(* Logix 5000 project; controller FRC_CC_2020 vendor 1 type 14 code 150 rev 31.11; software revision 31.01; part 2 of 4 *)
(* tags used below, declared in another part *)
   BlueESTOP1 : ALIAS FOR Blue_Driver_station:I.Data.14;
   BlueESTOP2 : ALIAS FOR Blue_Driver_station:I.Data.12;
   BlueESTOP3 : ALIAS FOR Blue_Driver_station:I.Data.10;
   Connection : INT;
   Field_Reset_Green : BOOL;
   FieldESTOP : BOOL;
   FieldESTOPButton : ALIAS FOR Local:1:I.Data.0;
   MatchReset : BOOL;
   MatchSYNC : TIMER;
   MBTI_Change_Log_MSG : MESSAGE;
   MBTI_Conn_Acc_Timeout_MSG : MESSAGE;
   MBTI_Conn_Accept_MSG : MESSAGE;
   MBTI_ConnectionsLastErrors : DINT;
   MBTI_Create_Sock_MSG : MESSAGE;
   MBTI_Delete_All_MSG : MESSAGE;
   MBTI_Instance : DINT;
   MBTI_Read_Data_MSG_00 : MESSAGE;
   MBTI_Read_Data_MSG_01 : MESSAGE;
   MBTI_Read_Data_MSG_02 : MESSAGE;
   MBTI_Read_Data_MSG_03 : MESSAGE;
   MBTI_Read_Data_MSG_04 : MESSAGE;
   MBTI_Read_Data_MSG_05 : MESSAGE;
   MBTI_Read_Data_MSG_06 : MESSAGE;
   MBTI_Read_Data_MSG_07 : MESSAGE;
   MBTI_Read_Data_MSG_08 : MESSAGE;
   MBTI_Read_Data_MSG_09 : MESSAGE;
   MBTI_Read_Done : BOOL[32];
   MBTI_Read_Resp : READ_RESP_STR[10];
   MBTI_RW_Inactivity_MSG : MESSAGE;
   MBTI_Sock_Accept_Resp : AcceptResponse;
   MBTI_Total_Open : INT;
   MBTI_Total_Open_MSG : MESSAGE;
   MBTI_Write_Data_MSG_00 : MESSAGE;
   MBTI_Write_Data_MSG_01 : MESSAGE;
   MBTI_Write_Data_MSG_02 : MESSAGE;
   MBTI_Write_Data_MSG_03 : MESSAGE;
   MBTI_Write_Data_MSG_04 : MESSAGE;
   MBTI_Write_Data_MSG_05 : MESSAGE;
   MBTI_Write_Data_MSG_06 : MESSAGE;
   MBTI_Write_Data_MSG_07 : MESSAGE;
   MBTI_Write_Data_MSG_08 : MESSAGE;
   MBTI_Write_Data_MSG_09 : MESSAGE;
   MBTI_Write_Data_Out : WRT_DATA[10];
   MBTU_Enable_MBTCP : BOOL;
   MBTU_EnetModulePort : STRING;
   MBTU_Log_Enable : DINT;
   MBTU_MB_0xx : BOOL[256];
   MBTU_MB_1xx : BOOL[256];
   MBTU_MB_3xx : INT[1000];
   MBTU_MB_4xx : INT[100];
   RedESTOP1 : ALIAS FOR Red_Driver_station:I.Data.14;
   RedESTOP2 : ALIAS FOR Red_Driver_station:I.Data.12;
   RedESTOP3 : ALIAS FOR Red_Driver_station:I.Data.10;
   SL_1 : BOOL;
   SL_2 : BOOL;
   SL_3 : BOOL;
   SL_B : BOOL;
   Stack_Light_Green : ALIAS FOR Local:1:O.Data.4;
   Watchdog : BOOL;
(* MainProgram, continued *)

ROUTINE Tag_Converter_Static   (* ladder *)
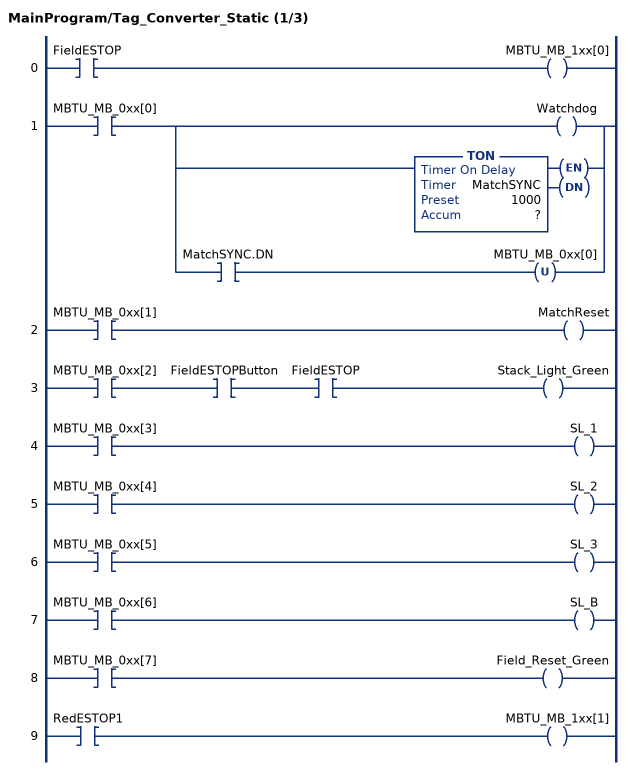
   0: XIC(FieldESTOP)OTE(MBTU_MB_1xx[0]);
   1: XIC(MBTU_MB_0xx[0])[OTE(Watchdog) ,TON(MatchSYNC,?,?) ,XIC(MatchSYNC.DN) OTU(MBTU_MB_0xx[0]) ];
   2: XIC(MBTU_MB_0xx[1])OTE(MatchReset);
   3: XIC(MBTU_MB_0xx[2])XIC(FieldESTOPButton)XIC(FieldESTOP)OTE(Stack_Light_Green);
   4: XIC(MBTU_MB_0xx[3])OTE(SL_1);
   5: XIC(MBTU_MB_0xx[4])OTE(SL_2);
   6: XIC(MBTU_MB_0xx[5])OTE(SL_3);
   7: XIC(MBTU_MB_0xx[6])OTE(SL_B);
   8: XIC(MBTU_MB_0xx[7])OTE(Field_Reset_Green);
   9: XIC(RedESTOP1)OTE(MBTU_MB_1xx[1]);
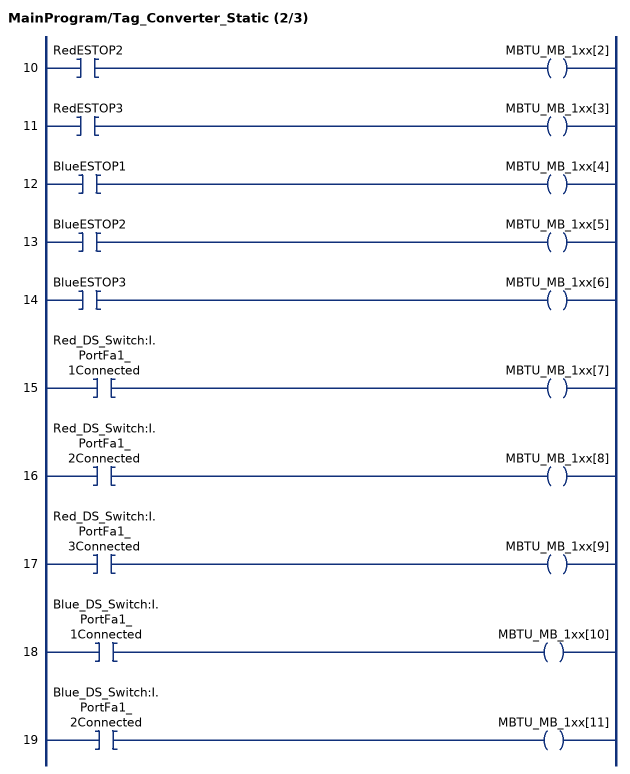
   10: XIC(RedESTOP2)OTE(MBTU_MB_1xx[2]);
   11: XIC(RedESTOP3)OTE(MBTU_MB_1xx[3]);
   12: XIC(BlueESTOP1)OTE(MBTU_MB_1xx[4]);
   13: XIC(BlueESTOP2)OTE(MBTU_MB_1xx[5]);
   14: XIC(BlueESTOP3)OTE(MBTU_MB_1xx[6]);
   15: XIC(Red_DS_Switch:I.PortFa1_1Connected)OTE(MBTU_MB_1xx[7]);
   16: XIC(Red_DS_Switch:I.PortFa1_2Connected)OTE(MBTU_MB_1xx[8]);
   17: XIC(Red_DS_Switch:I.PortFa1_3Connected)OTE(MBTU_MB_1xx[9]);
   18: XIC(Blue_DS_Switch:I.PortFa1_1Connected)OTE(MBTU_MB_1xx[10]);
   19: XIC(Blue_DS_Switch:I.PortFa1_2Connected)OTE(MBTU_MB_1xx[11]);
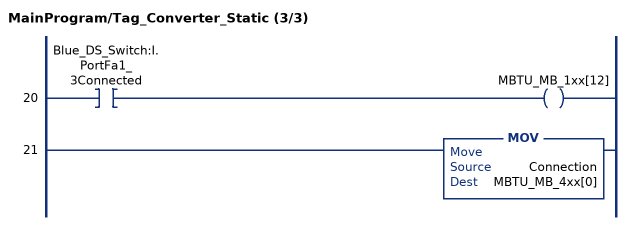
   20: XIC(Blue_DS_Switch:I.PortFa1_3Connected)OTE(MBTU_MB_1xx[12]);
   21: MOV(Connection,MBTU_MB_4xx[0]);
END_ROUTINE
END_PROGRAM

PROGRAM ModbusSlaveTCP   (* main routine Modbus_TCP_Slave *)
VAR
   Additional_len : INT := 6;
   Additional_len_read : INT := 12;
   buff_bit_index : DINT := 1;
   buff_byte_index : DINT := 3;
   CMD_END : DINT := 20;
   CMD_IN : DINT := 3;
   CMD_LEN : DINT := 21;
   CMD_LEN1 : INT := 42;
   CMD_LEN2 : INT := 45;
   CMD_START : DINT;
   Coil_Byte_Count : DINT := 3;
   coil_wr_index : DINT := 18;
   Conn_Open : BOOL[32] := ([0] := 1, [10] := 1, [11] := 1, [12] := 1, [13] := 1, [14] := 1, [15] := 1, [16] := 1, [17] := 1, [18] := 1, [19] := 1);
   Data_Received : BOOL;
   EX_CMD : INT := 144;
   EX_CODE : INT := 2;
   Found : BOOL := 1;
   INT_DATA_IN : INT := 11520;
   INT_IN : INT := 3;
   INT_STR_OUT : STRING := '$00$06';
   Listen_Retry_Tmr : TIMER := (PRE := 20);
   Listen_Socket_Lost : BOOL;
   Log_Old : DINT := 255;
   Main_Read_Buffer : STR_4096[20];
   mb_bit_index : DINT := 17;
   MB_Resp_Data : STR_462 := '$0F$00$00$00$13';
   MB_TMP_INT : INT := -5632;
   Modbus_Byte_cnt : INT := 240;
   Modbus_Bytes : DINT := 5;
   Modbus_CMD_Len : INT := 5376;
   Modbus_Cmd_String : STR_462 := '$03$00$00$00$15';
   Modbus_ID : STRING := '$A8$8D$00$00';
   Modbus_Packet : STR_462 := '$A8$CD$00$00$00$06$FF$03$00$00$00$15';
   Modbus_resp_Str : STR_462 := '$A8$CD$00$00$00-$FF$03*$00$0F$00$00$00$00$00$00$00$00$00$00$00$00$09$9C$03O$03$12$04f$02?$05I$08u$05$19$00$00$00$02$00$00$00$00$00$00$00$00';
   Modbus_Ret_CMD : STRING := '$03';
   Modbus_Ret_len : STRING := '$00$06';
   Modbus_Start : INT;
   Modbus_Unit : STRING := '$FF';
   Next_Write : BOOL[32];
   No_Open_Sockets : BOOL;
   Nothing : BOOL := 1;
   ONS : BOOL[64] := ([1] := 1, [2] := 1, [3] := 1, [4] := 1, [8] := 1);
   ONS_B : BOOL[32] := ([2] := 1, [3] := 1, [4] := 1, [5] := 1, [6] := 1, [7] := 1, [8] := 1, [9] := 1);
   ONS_ERR : BOOL[32] := ([1] := 1, [2] := 1, [3] := 1, [4] := 1, [5] := 1, [6] := 1, [7] := 1, [8] := 1, [9] := 1, [22] := 1, [23] := 1, [24] := 1, [25] := 1, [26] := 1, [27] := 1, [28] := 1, [29] := 1);
   RetryCreateSock : TIMER := (PRE := 2000);
   RG_4x_Pos : DINT := 21;
   RG_STR_TMP : STRING;
   RW_Instance : INT[20] := ([0] := 19547);
   RW_Select : DINT := 1;
   Startup_Timer : TIMER := (PRE := 1000, ACC := 1000, EN := 1, DN := 1);
   Str_Out : STR_1 := '$03';
   String_Pos : INT := 246;
   TestCntr : COUNTER := (PRE := 99999, ACC := 4733);
   testint : DINT;
   Valid : BOOL[32];
   Valid_CMD : BOOL[32] := ([2] := 1, [3] := 1);
   Valid_Command : BOOL;
   Valid_End : BOOL := 1;
   Valid_Len : BOOL := 1;
   Valid_Len_16 : BOOL;
   Valid_Start_Addr : BOOL := 1;
   Valid_Value_05 : BOOL;
   W_Log_Accept : ALIAS FOR MBTU_Log_Enable.2;
   W_Log_Attribute : ALIAS FOR MBTU_Log_Enable.6;
   W_Log_Create : ALIAS FOR MBTU_Log_Enable.0;
   W_Log_Delete : ALIAS FOR MBTU_Log_Enable.5;
   W_Log_Errors : ALIAS FOR MBTU_Log_Enable.7;
   W_Log_Open : ALIAS FOR MBTU_Log_Enable.1;
   W_Log_Read : ALIAS FOR MBTU_Log_Enable.3;
   W_Log_Write : ALIAS FOR MBTU_Log_Enable.4;
END_VAR

ROUTINE _SUB_0x_RD   (* ladder *)
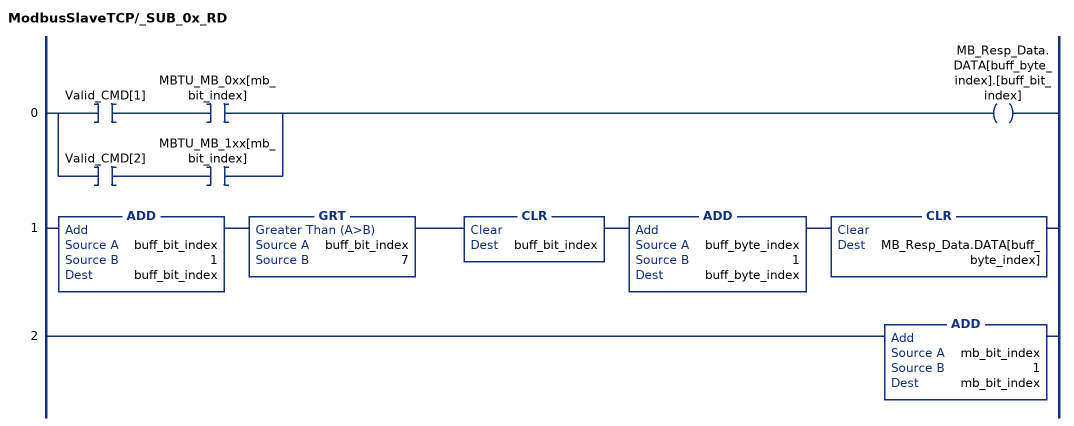
   0: [XIC(Valid_CMD[1]) XIC(MBTU_MB_0xx[mb_bit_index]) ,XIC(Valid_CMD[2]) XIC(MBTU_MB_1xx[mb_bit_index]) ]OTE(MB_Resp_Data.DATA[buff_byte_index].[buff_bit_index]);
   1: ADD(buff_bit_index,1,buff_bit_index)GRT(buff_bit_index,7)CLR(buff_bit_index)ADD(buff_byte_index,1,buff_byte_index)CLR(MB_Resp_Data.DATA[buff_byte_index]);
   2: ADD(mb_bit_index,1,mb_bit_index);
END_ROUTINE

ROUTINE _SUB_0x_WR   (* ladder *)
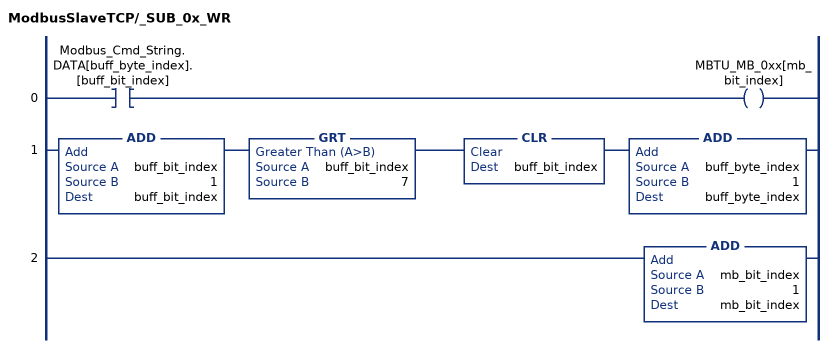
   0: XIC(Modbus_Cmd_String.DATA[buff_byte_index].[buff_bit_index])OTE(MBTU_MB_0xx[mb_bit_index]);
   1: ADD(buff_bit_index,1,buff_bit_index)GRT(buff_bit_index,7)CLR(buff_bit_index)ADD(buff_byte_index,1,buff_byte_index);
   2: ADD(mb_bit_index,1,mb_bit_index);
END_ROUTINE

ROUTINE _SUB_4x_RD   (* ladder *)
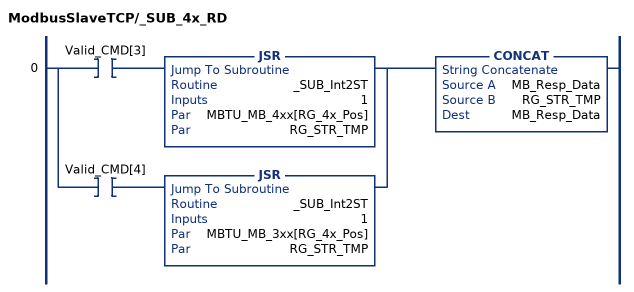
   0: [XIC(Valid_CMD[3]) JSR(_SUB_Int2ST,1,MBTU_MB_4xx[RG_4x_Pos],RG_STR_TMP) ,XIC(Valid_CMD[4]) JSR(_SUB_Int2ST,1,MBTU_MB_3xx[RG_4x_Pos],RG_STR_TMP) ]CONCAT(MB_Resp_Data,RG_STR_TMP,MB_Resp_Data);
END_ROUTINE

ROUTINE _SUB_4x_WR   (* ladder *)
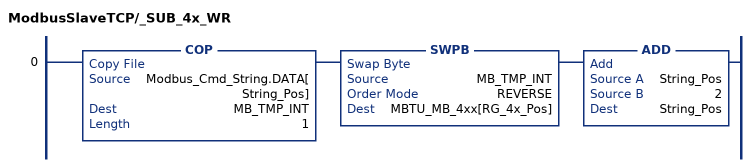
   0: COP(Modbus_Cmd_String.DATA[String_Pos],MB_TMP_INT,1)SWPB(MB_TMP_INT,REVERSE,MBTU_MB_4xx[RG_4x_Pos])ADD(String_Pos,2,String_Pos);
END_ROUTINE

ROUTINE _SUB_Byte2ST   (* ladder *)
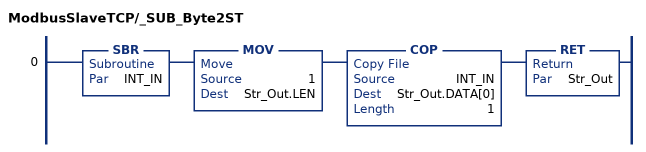
   0: SBR(INT_IN)MOV(1,Str_Out.LEN)COP(INT_IN,Str_Out.DATA[0],1)RET(Str_Out);
END_ROUTINE

ROUTINE _SUB_Int2ST   (* ladder *)
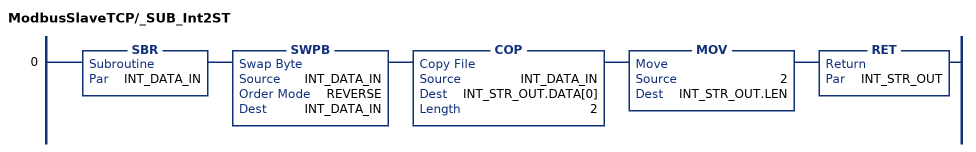
   0: SBR(INT_DATA_IN)SWPB(INT_DATA_IN,REVERSE,INT_DATA_IN)COP(INT_DATA_IN,INT_STR_OUT.DATA[0],2)MOV(2,INT_STR_OUT.LEN)RET(INT_STR_OUT);
END_ROUTINE

ROUTINE _SUB_SET_PATH   (* ladder *)
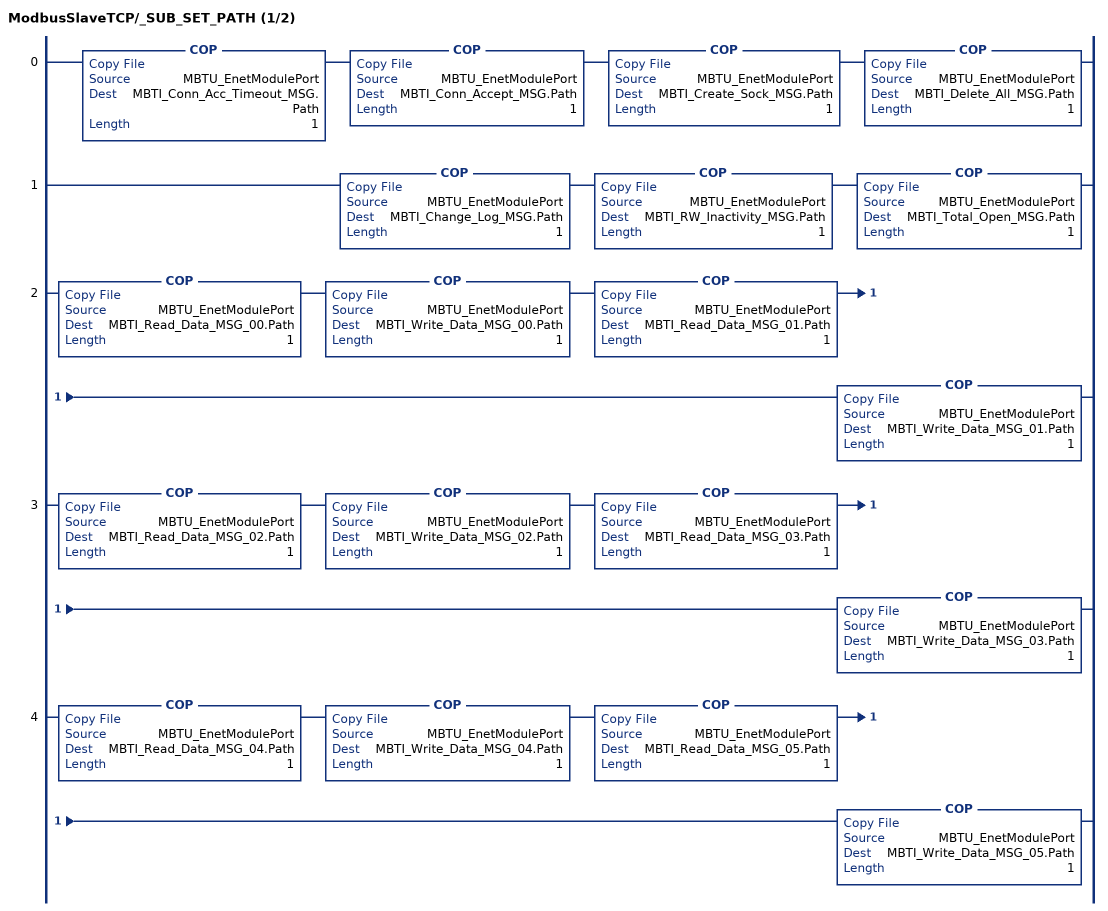
   0: COP(MBTU_EnetModulePort,MBTI_Conn_Acc_Timeout_MSG.Path,1)COP(MBTU_EnetModulePort,MBTI_Conn_Accept_MSG.Path,1)COP(MBTU_EnetModulePort,MBTI_Create_Sock_MSG.Path,1)COP(MBTU_EnetModulePort,MBTI_Delete_All_MSG.Path,1);
   1: COP(MBTU_EnetModulePort,MBTI_Change_Log_MSG.Path,1)COP(MBTU_EnetModulePort,MBTI_RW_Inactivity_MSG.Path,1)COP(MBTU_EnetModulePort,MBTI_Total_Open_MSG.Path,1);
   2: COP(MBTU_EnetModulePort,MBTI_Read_Data_MSG_00.Path,1)COP(MBTU_EnetModulePort,MBTI_Write_Data_MSG_00.Path,1)COP(MBTU_EnetModulePort,MBTI_Read_Data_MSG_01.Path,1)COP(MBTU_EnetModulePort,MBTI_Write_Data_MSG_01.Path,1);
   3: COP(MBTU_EnetModulePort,MBTI_Read_Data_MSG_02.Path,1)COP(MBTU_EnetModulePort,MBTI_Write_Data_MSG_02.Path,1)COP(MBTU_EnetModulePort,MBTI_Read_Data_MSG_03.Path,1)COP(MBTU_EnetModulePort,MBTI_Write_Data_MSG_03.Path,1);
   4: COP(MBTU_EnetModulePort,MBTI_Read_Data_MSG_04.Path,1)COP(MBTU_EnetModulePort,MBTI_Write_Data_MSG_04.Path,1)COP(MBTU_EnetModulePort,MBTI_Read_Data_MSG_05.Path,1)COP(MBTU_EnetModulePort,MBTI_Write_Data_MSG_05.Path,1);
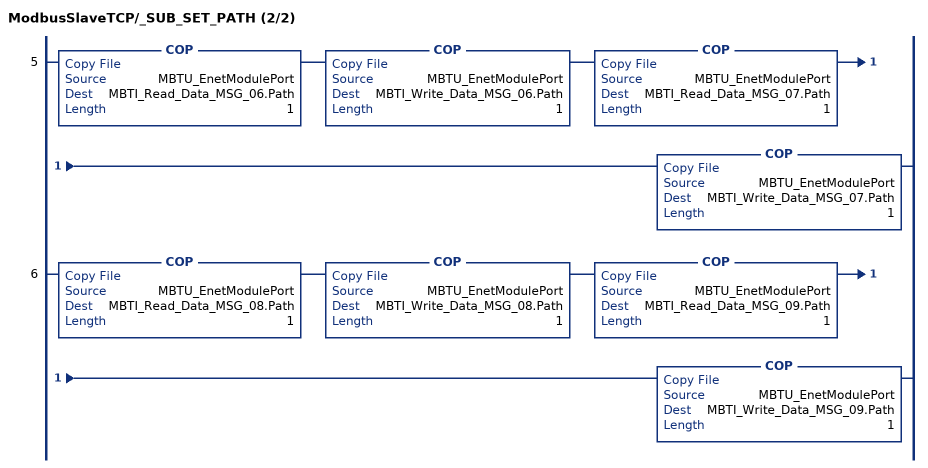
   5: COP(MBTU_EnetModulePort,MBTI_Read_Data_MSG_06.Path,1)COP(MBTU_EnetModulePort,MBTI_Write_Data_MSG_06.Path,1)COP(MBTU_EnetModulePort,MBTI_Read_Data_MSG_07.Path,1)COP(MBTU_EnetModulePort,MBTI_Write_Data_MSG_07.Path,1);
   6: COP(MBTU_EnetModulePort,MBTI_Read_Data_MSG_08.Path,1)COP(MBTU_EnetModulePort,MBTI_Write_Data_MSG_08.Path,1)COP(MBTU_EnetModulePort,MBTI_Read_Data_MSG_09.Path,1)COP(MBTU_EnetModulePort,MBTI_Write_Data_MSG_09.Path,1);
END_ROUTINE

ROUTINE Modbus_TCP_Slave   (* ladder *)
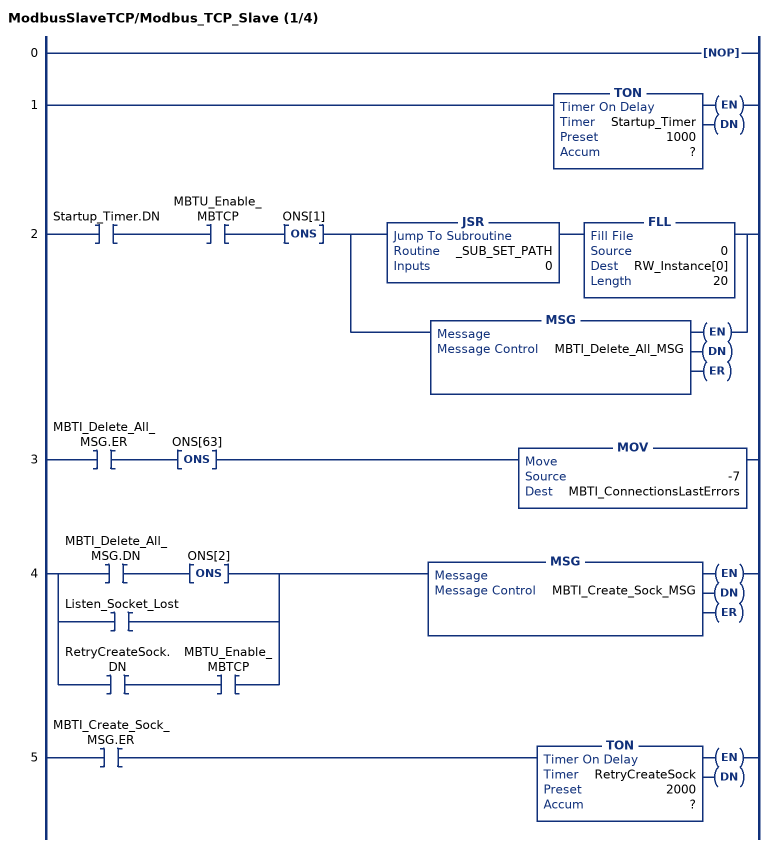
   0: NOP();
   1: TON(Startup_Timer,?,?);
   2: XIC(Startup_Timer.DN)XIC(MBTU_Enable_MBTCP)ONS(ONS[1])[JSR(_SUB_SET_PATH,0) FLL(0,RW_Instance[0],20) ,MSG(MBTI_Delete_All_MSG) ];
   3: XIC(MBTI_Delete_All_MSG.ER)ONS(ONS[63])MOV(-7,MBTI_ConnectionsLastErrors);
   4: [XIC(MBTI_Delete_All_MSG.DN) ONS(ONS[2]) ,XIC(Listen_Socket_Lost) ,XIC(RetryCreateSock.DN) XIC(MBTU_Enable_MBTCP) ]MSG(MBTI_Create_Sock_MSG);
   5: XIC(MBTI_Create_Sock_MSG.ER)TON(RetryCreateSock,?,?);
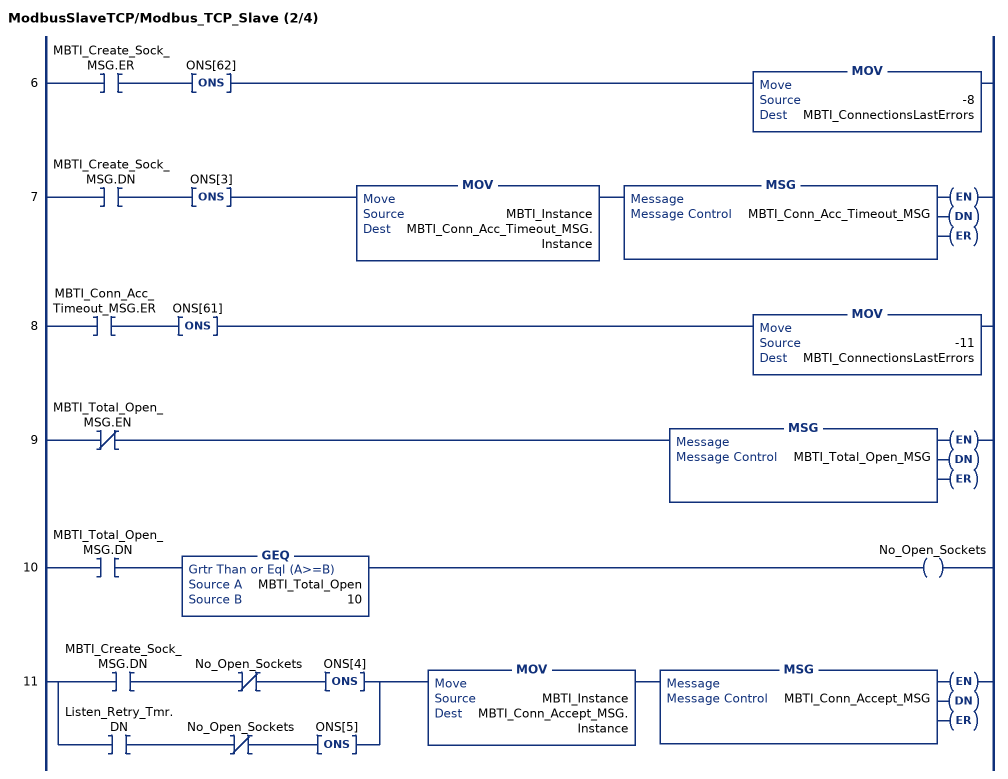
   6: XIC(MBTI_Create_Sock_MSG.ER)ONS(ONS[62])MOV(-8,MBTI_ConnectionsLastErrors);
   7: XIC(MBTI_Create_Sock_MSG.DN)ONS(ONS[3])MOV(MBTI_Instance,MBTI_Conn_Acc_Timeout_MSG.Instance)MSG(MBTI_Conn_Acc_Timeout_MSG);
   8: XIC(MBTI_Conn_Acc_Timeout_MSG.ER)ONS(ONS[61])MOV(-11,MBTI_ConnectionsLastErrors);
   9: XIO(MBTI_Total_Open_MSG.EN)MSG(MBTI_Total_Open_MSG);
   10: XIC(MBTI_Total_Open_MSG.DN)GEQ(MBTI_Total_Open,10)OTE(No_Open_Sockets);
   11: [XIC(MBTI_Create_Sock_MSG.DN) XIO(No_Open_Sockets) ONS(ONS[4]) ,XIC(Listen_Retry_Tmr.DN) XIO(No_Open_Sockets) ONS(ONS[5]) ]MOV(MBTI_Instance,MBTI_Conn_Accept_MSG.Instance)MSG(MBTI_Conn_Accept_MSG);
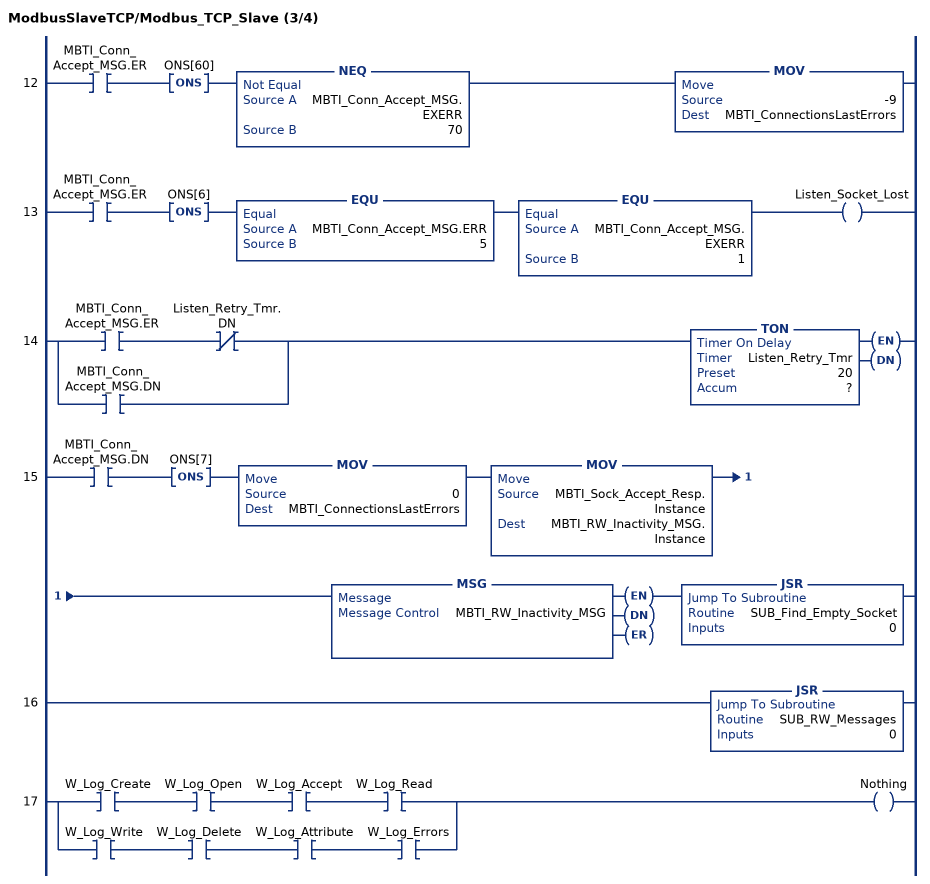
   12: XIC(MBTI_Conn_Accept_MSG.ER)ONS(ONS[60])NEQ(MBTI_Conn_Accept_MSG.EXERR,70)MOV(-9,MBTI_ConnectionsLastErrors);
   13: XIC(MBTI_Conn_Accept_MSG.ER)ONS(ONS[6])EQU(MBTI_Conn_Accept_MSG.ERR,5)EQU(MBTI_Conn_Accept_MSG.EXERR,1)OTE(Listen_Socket_Lost);
   14: [XIC(MBTI_Conn_Accept_MSG.ER) XIO(Listen_Retry_Tmr.DN) ,XIC(MBTI_Conn_Accept_MSG.DN) ]TON(Listen_Retry_Tmr,?,?);
   15: XIC(MBTI_Conn_Accept_MSG.DN)ONS(ONS[7])MOV(0,MBTI_ConnectionsLastErrors)MOV(MBTI_Sock_Accept_Resp.Instance,MBTI_RW_Inactivity_MSG.Instance)MSG(MBTI_RW_Inactivity_MSG)JSR(SUB_Find_Empty_Socket,0);
   16: JSR(SUB_RW_Messages,0);
   17: [XIC(W_Log_Create) XIC(W_Log_Open) XIC(W_Log_Accept) XIC(W_Log_Read) ,XIC(W_Log_Write) XIC(W_Log_Delete) XIC(W_Log_Attribute) XIC(W_Log_Errors) ]OTE(Nothing);
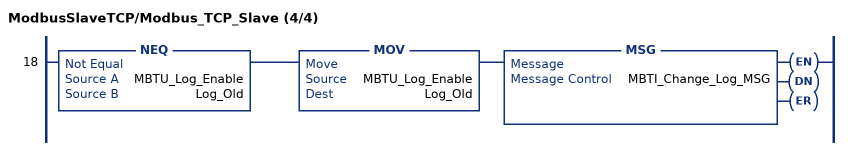
   18: NEQ(MBTU_Log_Enable,Log_Old)MOV(MBTU_Log_Enable,Log_Old)MSG(MBTI_Change_Log_MSG);
END_ROUTINE

ROUTINE Packet_Processing   (* ladder *)
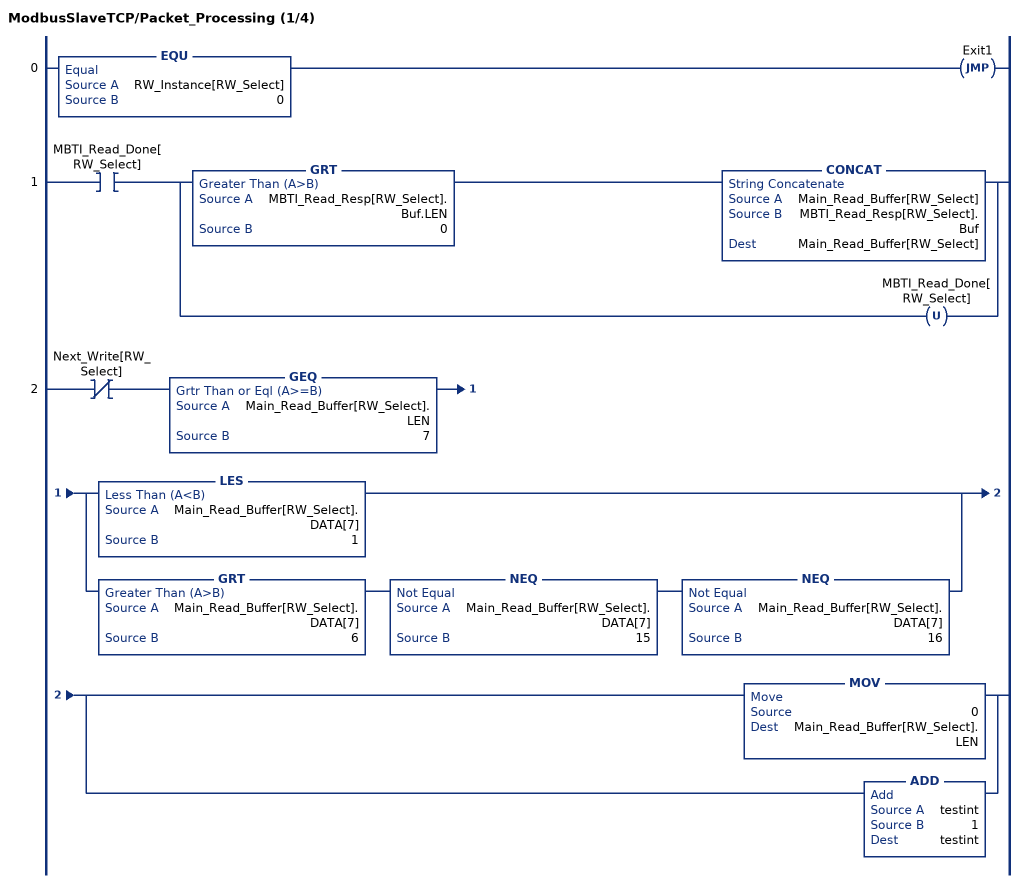
   0: EQU(RW_Instance[RW_Select],0)JMP(Exit1);
   1: XIC(MBTI_Read_Done[RW_Select])[GRT(MBTI_Read_Resp[RW_Select].Buf.LEN,0) CONCAT(Main_Read_Buffer[RW_Select],MBTI_Read_Resp[RW_Select].Buf,Main_Read_Buffer[RW_Select]) ,OTU(MBTI_Read_Done[RW_Select]) ];
   2: XIO(Next_Write[RW_Select])GEQ(Main_Read_Buffer[RW_Select].LEN,7)[LES(Main_Read_Buffer[RW_Select].DATA[7],1) ,GRT(Main_Read_Buffer[RW_Select].DATA[7],6) NEQ(Main_Read_Buffer[RW_Select].DATA[7],15) NEQ(Main_Read_Buffer[RW_Select].DATA[7],16) ][MOV(0,Main_Read_Buffer[RW_Select].LEN) ,ADD(testint,1,testint) ];
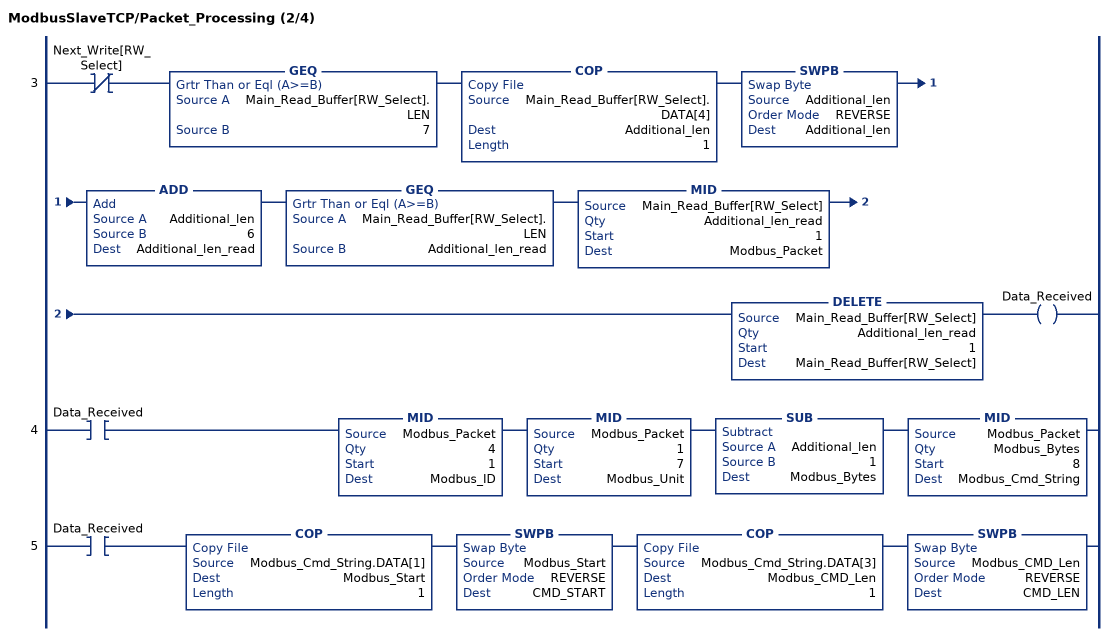
   3: XIO(Next_Write[RW_Select])GEQ(Main_Read_Buffer[RW_Select].LEN,7)COP(Main_Read_Buffer[RW_Select].DATA[4],Additional_len,1)SWPB(Additional_len,REVERSE,Additional_len)ADD(Additional_len,6,Additional_len_read)GEQ(Main_Read_Buffer[RW_Select].LEN,Additional_len_read)MID(Main_Read_Buffer[RW_Select],Additional_len_read,1,Modbus_Packet)DELETE(Main_Read_Buffer[RW_Select],Additional_len_read,1,Main_Read_Buffer[RW_Select])OTE(Data_Received);
   4: XIC(Data_Received)MID(Modbus_Packet,4,1,Modbus_ID)MID(Modbus_Packet,1,7,Modbus_Unit)SUB(Additional_len,1,Modbus_Bytes)MID(Modbus_Packet,Modbus_Bytes,8,Modbus_Cmd_String);
   5: XIC(Data_Received)COP(Modbus_Cmd_String.DATA[1],Modbus_Start,1)SWPB(Modbus_Start,REVERSE,CMD_START)COP(Modbus_Cmd_String.DATA[3],Modbus_CMD_Len,1)SWPB(Modbus_CMD_Len,REVERSE,CMD_LEN);
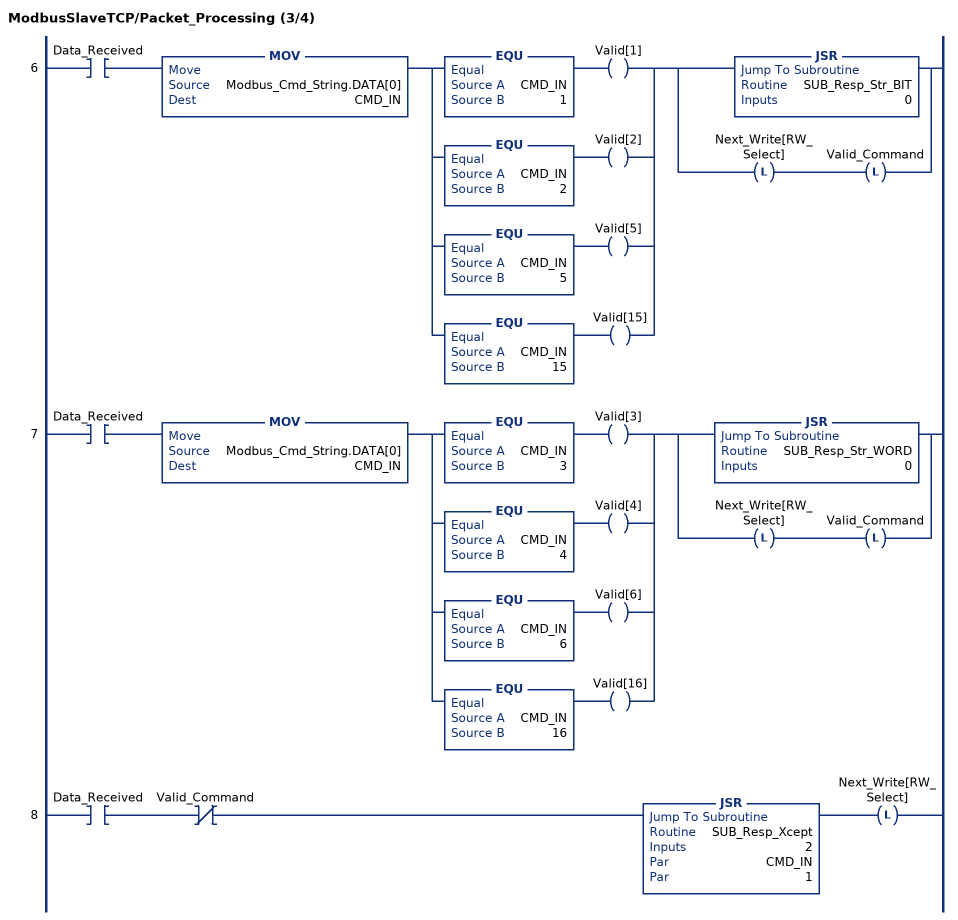
   6: XIC(Data_Received)MOV(Modbus_Cmd_String.DATA[0],CMD_IN)[EQU(CMD_IN,1) OTE(Valid[1]) ,EQU(CMD_IN,2) OTE(Valid[2]) ,EQU(CMD_IN,5) OTE(Valid[5]) ,EQU(CMD_IN,15) OTE(Valid[15]) ][JSR(SUB_Resp_Str_BIT,0) ,OTL(Next_Write[RW_Select]) OTL(Valid_Command) ];
   7: XIC(Data_Received)MOV(Modbus_Cmd_String.DATA[0],CMD_IN)[EQU(CMD_IN,3) OTE(Valid[3]) ,EQU(CMD_IN,4) OTE(Valid[4]) ,EQU(CMD_IN,6) OTE(Valid[6]) ,EQU(CMD_IN,16) OTE(Valid[16]) ][JSR(SUB_Resp_Str_WORD,0) ,OTL(Next_Write[RW_Select]) OTL(Valid_Command) ];
   8: XIC(Data_Received)XIO(Valid_Command)JSR(SUB_Resp_Xcept,2,CMD_IN,1)OTL(Next_Write[RW_Select]);
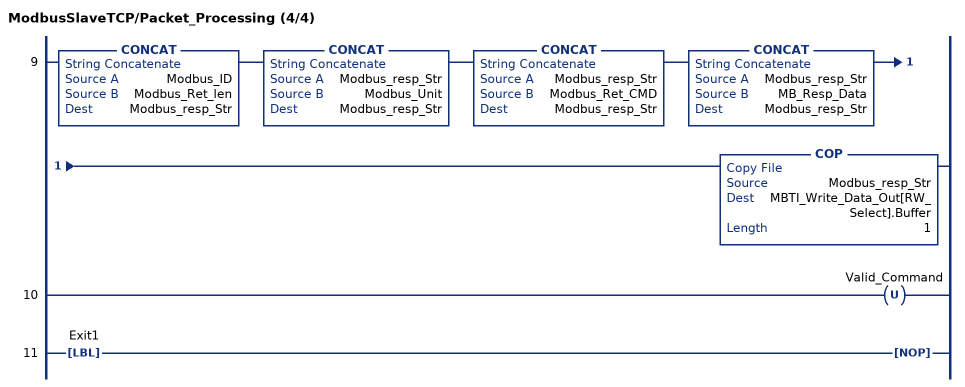
   9: CONCAT(Modbus_ID,Modbus_Ret_len,Modbus_resp_Str)CONCAT(Modbus_resp_Str,Modbus_Unit,Modbus_resp_Str)CONCAT(Modbus_resp_Str,Modbus_Ret_CMD,Modbus_resp_Str)CONCAT(Modbus_resp_Str,MB_Resp_Data,Modbus_resp_Str)COP(Modbus_resp_Str,MBTI_Write_Data_Out[RW_Select].Buffer,1);
   10: OTU(Valid_Command);
   11: LBL(Exit1)NOP();
END_ROUTINE
